(* CODESYS project Connect with TSR.project

Project tree, tasks and I/O mapping:
  XV100 : XV100, Eaton Automation, version 3.5.3.0
    application Application
      libraries: Standard, 3.5.2.0 (System); CAA SerialCom, 3.5.3.0 (CAA Technical Workgroup); TSR Libary, 0.1 (Eaton Automation)
      task Task (cyclic, interval t#10ms, priority 1) calls MAIN
      Symbols
      program MAIN [ST]: A4_End, A3_Auswerten, A0_Start, A2_Progress_Wait, A1_Progress, B100_Error
*)

// XV100/Application/MAIN
PROGRAM MAIN
VAR
//FB EINGANGS VAR
xEXecute				:BOOL;		//Startbedingung für den FB.
iCom					:INT;		//Die Nummer des Com Ports.
//FB AUSGANGS VAR
xBusy					:BOOL;		//Das Busy bit.
xDone					:BOOL;		//Ist 1 wenn FB fertig ist.
wState					:WORD;		//Der ENUM Wert für die ENUM Tabelle.
xError					:BOOL;		//Ist 1 wenn es einen Error gab.

//INTERNE VAR
LTi_Zustand				:INT;		//Der Zustand.

//TIMER
FB_Timer				:TON;			//Timer Init
TSR_Com: 				TSR_Com;
END_VAR

//Parameters
VAR CONSTANT
LTt_WaitTimeout		:TIME := T#2S;		//der Timout Timer.

END_VAR

CASE LTi_Zustand OF
	0:
		A0_Start();					//Prüfe die Startbedingungen 
	1:
		A1_Progress();				//Starte den Prozess.
	2:
		A2_Progress_Wait();			//Warte auf den FB TSR Com
	3:
		A3_Auswerten();				//Werte das Egebniss aus.
	4:
		A4_End();					//Warte auf Execute
	100:
		B100_Error();				//Nur wenn ein Error gab.
END_CASE

TSR_Com();

ACTION A4_End:
xBusy := 0;							//Alles zurücksetzten
xDone := 1;
IF xExecute = 0 THEN				//Warten bis der User Zurückgesetzt hat.
	xDone := 0;
	LTi_Zustand := 0;
	TSR_Com.xEXecute := 0;
END_IF
END_ACTION

ACTION A3_Auswerten:
IF TSR_Com.stReceivedData = '!' THEN		//Wenn der TSR reagiert.
	LTi_Zustand := 4;						//Gehe zum letzten Zustand.
ELSE										//Ansonten ist es ein Fehler.
	LTi_Zustand := 100;	
	wState := 8;							//Gib beim State die ENUM Zahl an.
END_IF
END_ACTION

ACTION A0_Start:
IF xExecute THEN			//Prüfe Startbedinung.
	xBusy := 1;				//Setze Busy.
	LTi_Zustand := 1;	//Gehe direkt zum Schritt wo der Com Port geöffnet wird.
END_IF
END_ACTION

ACTION A2_Progress_Wait:
IF TSR_Com.xDone THEN											//Wenn der Port offen
	FB_Timer.IN := 0;					//Timer Zurücksetzten.
	LTi_Zustand := 3;					//Gehe in den Sende Schritt
ELSE
	IF TSR_Com.xError THEN				//Wenn es einen Error bei Com Port öffnen gab.
		FB_Timer.IN := 0;					//Timer Zurücksetzten.
		LTi_Zustand := 100;					//In den Error Zustand gehen.
		wState := TSR_Com.wState;			//Den ENUM Wert Error angeben.
	ELSE
		IF FB_Timer.Q THEN						//Wenn der Timer Abgelaufen ist.
			LTi_Zustand := 100;					//In den Error Zustand gehen.
			wState := 7;						//Den ENUM Wert Error angeben.
			FB_Timer.IN := 0;
		END_IF
	END_IF
FB_Timer(IN := 1, PT:= LTt_WaitTimeout);
END_IF

FB_Timer();								//Rufe Timer auf
END_ACTION

ACTION A1_Progress:
TSR_Com(						//TSR Com Aufrufen und Daten übergeben.
	xEXecute	:=	1 , 
	iCom		:= 	iCom, 
	stSendData	:= 	'?',  );
LTi_Zustand := 2;				//In den nächsten Zustand Wechseln.
END_ACTION

ACTION B100_Error:
xBusy := 0;							//Alles zurücksetzten
xError := 1;
IF xExecute = 0 THEN				//Wartem bis der User das xExecute zurückgesetzt hat.
	xError := 0;
	LTi_Zustand := 0;
	wState := 0;
	TSR_Com.xEXecute := 0;
END_IF
END_ACTION

END_PROGRAM
